PROGRAM VGC1
VAR
END_VAR

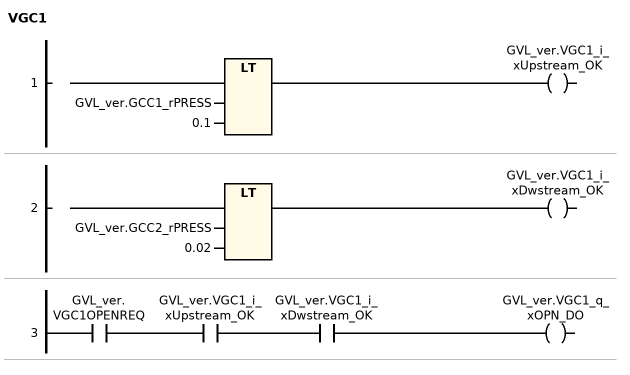
// NETWORK 1
GVL_ver.VGC1_i_xUpstream_OK := GVL_ver.GCC1_rPRESS < 0.1;

// NETWORK 2
GVL_ver.VGC1_i_xDwstream_OK := GVL_ver.GCC2_rPRESS < 0.02;

// NETWORK 3
GVL_ver.VGC1_q_xOPN_DO := GVL_ver.VGC1OPENREQ AND GVL_ver.VGC1_i_xUpstream_OK AND GVL_ver.VGC1_i_xDwstream_OK;

END_PROGRAM

(* stored: Version 1.1.0.1, ProductVersion 3.1.4022.3
   POU VGC1: Id {827b8fce-a213-4f84-a2b2-b57f49854814}, SpecialFunc None *)
